(* Check if a certain test in the current suite is finished *)
FUNCTION IS_TEST_FINISHED : BOOL
VAR_INPUT
    TestName : Tc2_System.T_MaxString;
END_VAR
VAR
    Counter : UINT;
    CurrentTest : FB_Test;
END_VAR

TestName := F_LTrim(in := F_RTrim(in := TestName));

IS_TEST_FINISHED := FALSE;

FOR Counter := 1 TO GVL_TcUnit.CurrentTestSuiteBeingCalled^.GetNumberOfTests() BY 1 DO
    CurrentTest := GVL_TcUnit.CurrentTestSuiteBeingCalled^.Tests[Counter];
    IF CurrentTest.TestName = TestName THEN
        IS_TEST_FINISHED := CurrentTest.IsFinished();
        RETURN;
    END_IF
END_FOR

END_FUNCTION

(* stored: Version 1.1.0.1
   POU IS_TEST_FINISHED: Id {79206b95-49a5-42aa-8a6a-b089aa13b1fd}, SpecialFunc None *)
